{attribute 'qualified_only'}
{attribute 'strict'}
TYPE EStagePosition :
(
	Unknown := 0,
	Loading,
	Process
);
END_TYPE

(* stored: Version 1.1.0.1, ProductVersion 3.1.4024.12
   DUT EStagePosition: Id {687b209c-0a9c-4fe7-ab73-5eb3fcb6db93} *)
